TYPE STATUS_HMI :
STRUCT
	isMoving : BOOL;
	isMovingWithObject : BOOL;
	movingToPosition : INT;
	currentPosition : INT;
	currentPositionWithObject : INT;
	movingDirection : E_DIRECTION;
	hasObject : BOOL;
	alarm : BOOL;
	alarmText : STRING;
	undefined : BOOL;
END_STRUCT
END_TYPE

(* stored: Version 1.1.0.1, ProductVersion 3.1.4024.12
   DUT STATUS_HMI: Id {53bf5917-e8a8-4455-8e2e-715ee8c35218} *)
